// Mitsubishi GX Works2 project: LRI - Lógica OR   PLC: Q03UDV
// HelloWorld

PROGRAM MAIN
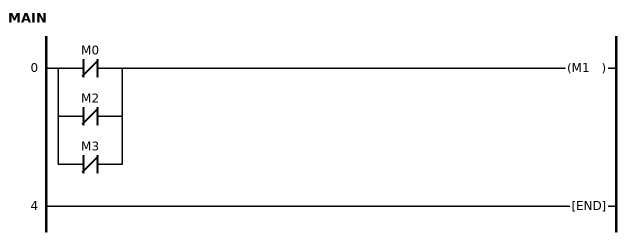
0     LDI     M0
      ORI     M2
      ORI     M3
      OUT     M1
4     END
END_PROGRAM
